{attribute 'GeneratedUsingTerminal: EK1100-0000-0018'}
{attribute addProperty BoxType "EK1100-0000-0018"}
{attribute addProperty Id "Beckhoff_ER7xxxEK1122Beckhoff_ER7xxxEK1122_D0247035686"}
{attribute addProperty CRC "1721877453"}
{attribute addProperty Size "686"}
TYPE Beckhoff_ER7xxx_66A1C3CD EXTENDS EK1100_AB5A9467 :
STRUCT
	{attribute addProperty Name "Beckhoff_ER7xxxEK1122"}
	Beckhoff_ER7xxxEK1122 : Beckhoff_ER7xxxEK1122_D0247035;
END_STRUCT
END_TYPE

(* stored: Version 1.2.0.0, ProductVersion 3.1.4024.9
   DUT Beckhoff_ER7xxx_66A1C3CD: Id {c345c412-5402-4ab1-ac21-b635c078a0f3} *)
